// TIA Portal V17 export
// export: Created 2023-02-14T02:49:24.9444304Z, ExportSetting WithDefaults, DisplayName Totally Integrated Automation Portal, DisplayVersion V17, DisplayName TIA Portal Openness, DisplayVersion V17, DisplayName TIA Portal Teamcenter Gateway, DisplayVersion V17, DisplayName TIA Portal Version Control Interface, DisplayVersion V17, DisplayName SINAMICS Startdrive Advanced, DisplayVersion V17, DisplayName SINAMICS Startdrive G130, G150, S120, S150, SINAMICS MV, S210, DisplayVersion V17, DisplayName SINAMICS Startdrive G110M, G120, G120C, G120D, G120P, G115D, DisplayVersion V17, DisplayName STEP 7 Professional, DisplayVersion V17, DisplayName STEP 7 Safety, DisplayVersion V17, DisplayName WinCC Professional, DisplayVersion V17
FUNCTION_BLOCK "IO Digital Blending"   // FB6, LAD
{ S7_Optimized_Access := 'FALSE' }
VERSION : 0.1
// stored: AutoNumber true, IsIECCheckEnabled false, SetENOAutomatically false, UDAEnableTagReadback false
   VAR_INPUT
      Init : Bool;
      Reset : Bool;
   END_VAR
   VAR
      "DRP-P22.01" { S7_SetPoint := 'True'} : "Digital";   // DRY RUN PROTECTION MONO PUMP P-22.01
      "DRP-P32.01" { S7_SetPoint := 'True'} : "Digital";   // DRY RUN PROTECTION MONO PUMP P-32.01
   END_VAR
BEGIN

REGION Network 1: DRP-P22.01
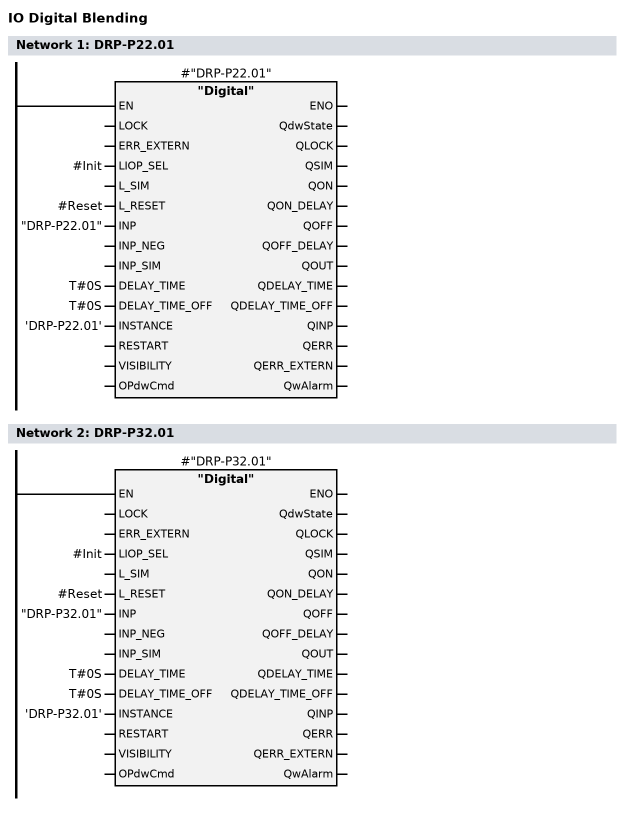
   RUNG wire#powerrail
      #"DRP-P22.01"(LOCK :=, ERR_EXTERN :=, LIOP_SEL := #Init, L_SIM :=, L_RESET := #Reset, INP := "DRP-P22.01", INP_NEG :=, INP_SIM :=, DELAY_TIME := T#0S, DELAY_TIME_OFF := T#0S, INSTANCE := 'DRP-P22.01', RESTART :=, VISIBILITY :=, OPdwCmd :=, QdwState =>, QLOCK =>, QSIM =>, QON =>, QON_DELAY =>, QOFF =>, QOFF_DELAY =>, QOUT =>, QDELAY_TIME =>, QDELAY_TIME_OFF =>, QINP =>, QERR =>, QERR_EXTERN =>, QwAlarm =>)
   END_RUNG
   // the same network as SCL:
   #"DRP-P22.01"(LIOP_SEL := #Init,   // "Digital"
                 L_RESET := #Reset,
                 INP := "DRP-P22.01",
                 DELAY_TIME := T#0S,
                 DELAY_TIME_OFF := T#0S,
                 INSTANCE := 'DRP-P22.01');
END_REGION

REGION Network 2: DRP-P32.01
   RUNG wire#powerrail
      #"DRP-P32.01"(LOCK :=, ERR_EXTERN :=, LIOP_SEL := #Init, L_SIM :=, L_RESET := #Reset, INP := "DRP-P32.01", INP_NEG :=, INP_SIM :=, DELAY_TIME := T#0S, DELAY_TIME_OFF := T#0S, INSTANCE := 'DRP-P32.01', RESTART :=, VISIBILITY :=, OPdwCmd :=, QdwState =>, QLOCK =>, QSIM =>, QON =>, QON_DELAY =>, QOFF =>, QOFF_DELAY =>, QOUT =>, QDELAY_TIME =>, QDELAY_TIME_OFF =>, QINP =>, QERR =>, QERR_EXTERN =>, QwAlarm =>)
   END_RUNG
   // the same network as SCL:
   #"DRP-P32.01"(LIOP_SEL := #Init,   // "Digital"
                 L_RESET := #Reset,
                 INP := "DRP-P32.01",
                 DELAY_TIME := T#0S,
                 DELAY_TIME_OFF := T#0S,
                 INSTANCE := 'DRP-P32.01');
END_REGION
END_FUNCTION_BLOCK
